FUNCTION_BLOCK SandboxContext EXTENDS TcoCore.TcoContext
VAR
    DataManager : TcoDataManager(THIS^);
	_state : INT;
END_VAR

(*~
	<docu>
		<summary>
			Main method of the TcoContext. This is the entry point of any control logic that belongs to this context. 
			The call of this method is ensured by calling the <c>InstanceName.Run()</c> method, and it must not be called explicitly.
			This method is abstract, and it must be overridden in derived block.
		</summary>
	</docu>
~*)
METHOD PROTECTED  Main
VAR
	recordId_1 : STRING;
	recordId_2 : STRING;
END_VAR
DataManager.Messenger.Build().Append('Entering data managed cyclic execution').As().AsDebug();
DataManager();

Context.Environment.Messaging.MessageDigestMethod := eMessageDigestMethod.CRC32;
Context.Environment.Messaging.MessengerLoggingMethod := eMessengerLogMethod.OnEventRisen;

recordId_1 := 'scoundrel';
recordId_2 := 'knight';

CASE _state OF
	0:
		IF(DataManager.Exists(recordId_1).Done) THEN
			IF(DataManager.Exists(recordId_1).Exists) THEN
				IF(DataManager.Delete(recordId_1).Done) THEN
					_state := 5;
				END_IF
			ELSE
				_state := 5;
			END_IF
		END_IF
	5:
		IF(DataManager.Exists(recordId_2).Done) THEN
			IF(DataManager.Exists(recordId_2).Exists) THEN
				IF(DataManager.Delete(recordId_2).Done) THEN
					_state := 10;
				END_IF
			ELSE
				_state := 10;
			END_IF
		END_IF	
	10:

// <CreateCodeExample>	
		// Will create new entry into repository with data contained in the `_data` 
		IF(DataManager.Create(recordId_1).Done) THEN
			_state := 20;
		END_IF;
// </CreateCodeExample>
		
	20:
		DataManager.Data.sampleData.SampleInt := 33;
		DataManager.Data.sampleData.SampleString := 'Max';
		DataManager.Data.sampleData.SampleNestedStructure.SampleLREAL := 1;
		IF(DataManager.Update(recordId_1).Done) THEN
			_state := 30;
		END_IF;	
	30:
		DataManager.Data.sampleData.SampleInt := 44;
		DataManager.Data.sampleData.SampleString := 'Lewis';
		DataManager.Data.sampleData.SampleNestedStructure.SampleLREAL := 7;
		IF(DataManager.CreateOrUpdate(recordId_2).Done) THEN
			_state := 40;
		END_IF;	
	40:		
		IF(DataManager.Read(recordId_1).Done) THEN
			_state := 50;
		END_IF;					
END_CASE
END_METHOD

END_FUNCTION_BLOCK

(* stored: Version 1.1.0.1, ProductVersion 3.1.4024.9
   POU SandboxContext: Id {ed8218eb-5f5f-0973-2882-9b75bfb2ad4d}, SpecialFunc None
   Method Main: Id {3a03a89e-90f1-0a89-181b-0e6b67acc445} *)
